// Mitsubishi GX Works2 project: CJ   PLC: Q03UDV

PROGRAM MAIN
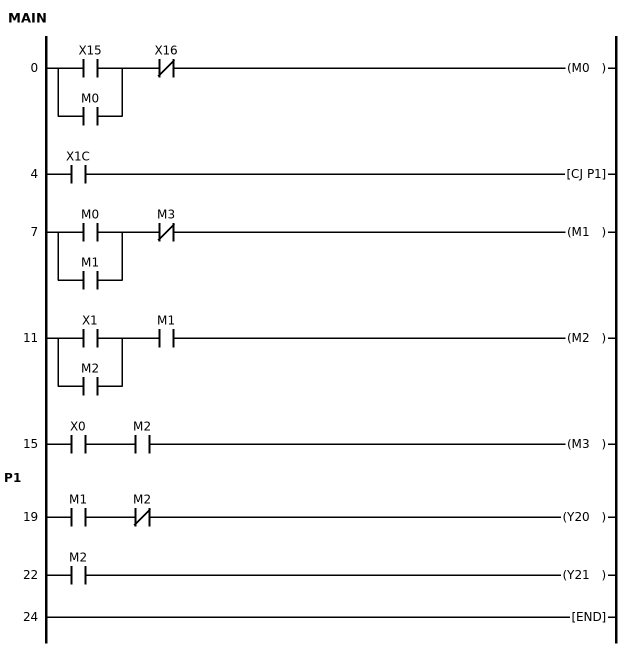
0     LD      X15
      OR      M0
      ANI     X16
      OUT     M0
4     LD      X1C
      CJ      P1
7     LD      M0
      OR      M1
      ANI     M3
      OUT     M1
11    LD      X1
      OR      M2
      AND     M1
      OUT     M2
15    LD      X0
      AND     M2
      OUT     M3
      P1
19    LD      M1
      ANI     M2
      OUT     Y20
22    LD      M2
      OUT     Y21
24    END
END_PROGRAM
